// SIMATIC S7-200 project (STEP 7-Micro/WIN), CPU 222 REL 02.01

SYMBOL_TABLE USER1
AI_1             AIW0     // TEMPERATURA DI SERVIZIO O RICIRCOLO
AI_2             AIW2     // TEMPERATURA CALDAIA
AI_3             AIW4     // TEMPERATURA AMBIENTE
AI_4             AIW6     // TEMPERATURA CIRCUITO DI RITORNO
M                AQW0     // COMANDO VALVOLA DI MISCELAZIONE
B1               Q0.0     // POMPA DI CIRCOLAZIONE LIVELLO 1
B2               Q0.1     // POMPA DI CIRCOLAZIONE LIVELLO 2
B3               Q0.2     // POMPA DI CIRCOLAZIONE LIVELLO 3
POMPA_2          Q0.3     // POMPA RISCALDAMENTO ACQUA USO DOMESTICO
BRC_1            Q0.4     // BRUCCIATORE LIVELLO 1
BRC_2            Q0.5     // BRUCCIATORE LIVELLO 2
BRC_3            Q1.0     // BRUCCIATORE LIVELLO 3
MIS_T_SERV       VD0      // MISURA TEMPERATURA DI SERVIZIO
MIS_T_CALDAIA    VD4      // MISURA TEMPERATURA CALDAIA
MIS_T_AMBIENTE   VD8      // MISURA TEMPERATURA AMBIENTE
MIS_T_RIT        VD12     // MISURA TEMPERATURA DI RITORNO
D_T              VD16     // DIFFERENZA DI TEMPERATURA FRA CALDAIA E RITORNO
END_SYMBOL_TABLE

ORGANIZATION_BLOCK MAIN:OB1
TITLE=DPS 210 IMPIANTO DI RISCALDAMENTO
BEGIN
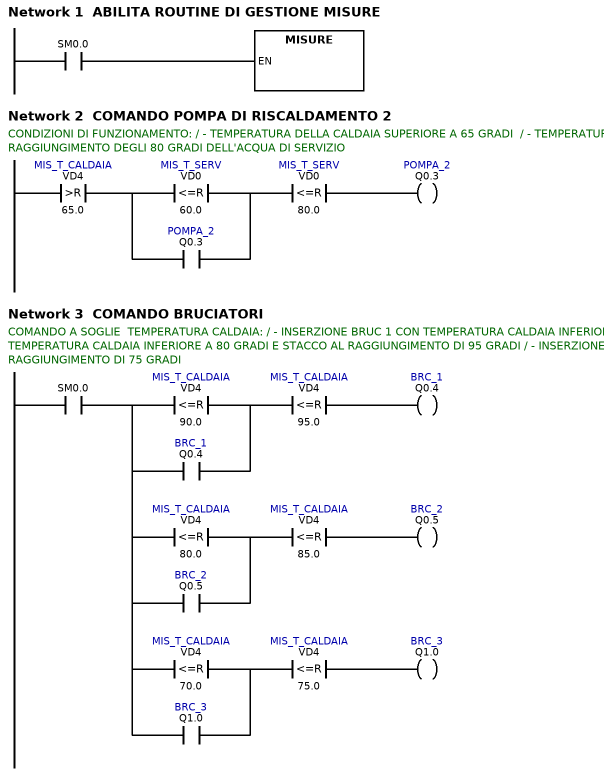
Network 1 // ABILITA ROUTINE DI GESTIONE MISURE
LD     SM0.0
CALL   MISURE:SBR1
Network 2 // COMANDO POMPA DI RISCALDAMENTO 2
// CONDIZIONI DI FUNZIONAMENTO:
// - TEMPERATURA DELLA CALDAIA SUPERIORE A 65 GRADI 
// - TEMPERATURA DI SERVIZIO INFERIORE A 60 GRADI
// PARTE LA POMPA DI CIRCOLAZIONE 2 FINO AL RAGGIUNGIMENTO DEGLI 80 GRADI DELL'ACQUA DI SERVIZIO
LDR>   MIS_T_CALDAIA:VD4, 65.0
LDR<=  MIS_T_SERV:VD0, 60.0
O      POMPA_2:Q0.3
ALD
AR<=   MIS_T_SERV:VD0, 80.0
=      POMPA_2:Q0.3
Network 3 // COMANDO BRUCIATORI
// COMANDO A SOGLIE  TEMPERATURA CALDAIA:
// - INSERZIONE BRUC 1 CON TEMPERATURA CALDAIA INFERIORE A 90 GRADI E STACCO AL RAGGIUNGIMENTO DI 95 GRADI
// - INSERZIONE BRUC 2 CON TEMPERATURA CALDAIA INFERIORE A 80 GRADI E STACCO AL RAGGIUNGIMENTO DI 95 GRADI
// - INSERZIONE BRUC 3 CON TEMPERATURA CALDAIA INFERIORE A 70 GRADI E STACCO AL RAGGIUNGIMENTO DI 75 GRADI
LD     SM0.0
LPS
LDR<=  MIS_T_CALDAIA:VD4, 90.0
O      BRC_1:Q0.4
ALD
AR<=   MIS_T_CALDAIA:VD4, 95.0
=      BRC_1:Q0.4
LRD
LDR<=  MIS_T_CALDAIA:VD4, 80.0
O      BRC_2:Q0.5
ALD
AR<=   MIS_T_CALDAIA:VD4, 85.0
=      BRC_2:Q0.5
LPP
LDR<=  MIS_T_CALDAIA:VD4, 70.0
O      BRC_3:Q1.0
ALD
AR<=   MIS_T_CALDAIA:VD4, 75.0
=      BRC_3:Q1.0
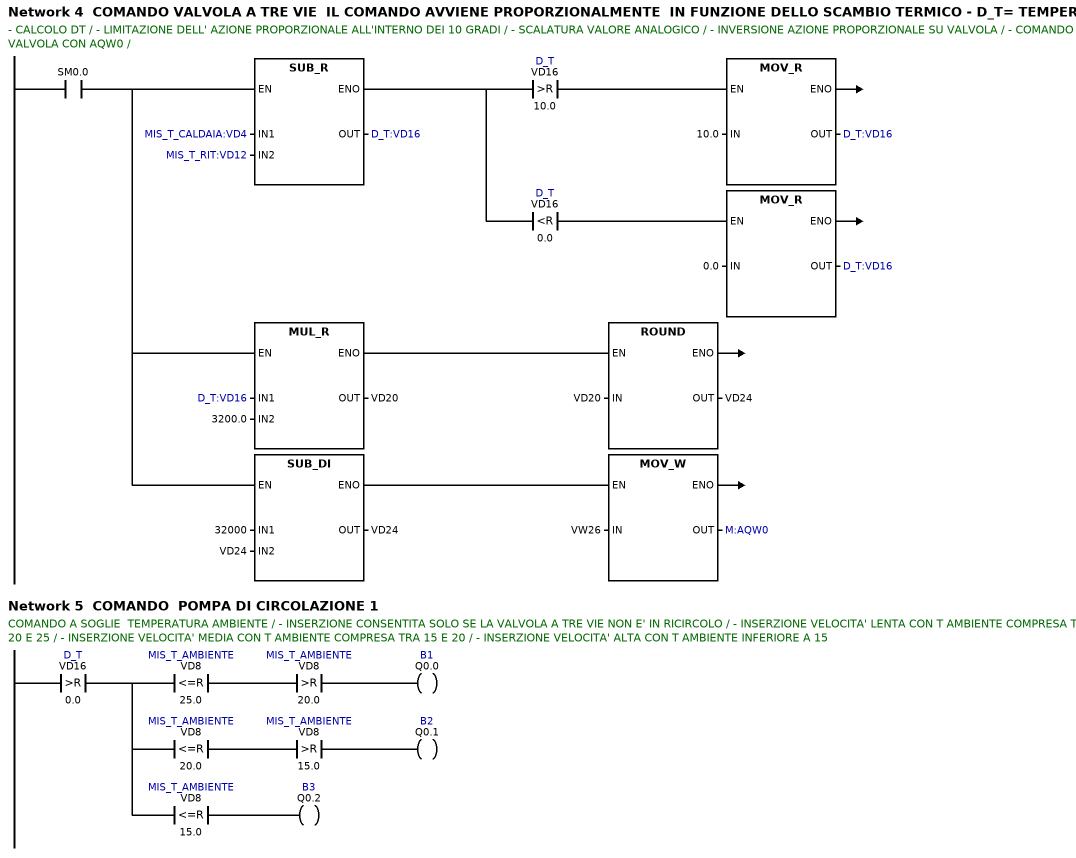
Network 4 // COMANDO VALVOLA A TRE VIE 
IL COMANDO AVVIENE PROPORZIONALMENTE  IN FUNZIONE DELLO SCAMBIO TERMICO
- D_T= TEMPERATURA CALDAIA - TEMPERATURA RITORNO
- D_T =0 VALVOLA TRE VIE IN RICIRCOLO
- D_T= 10 VALVOLA TRE VIE IN PIENA MANDATA
// - CALCOLO DT
// - LIMITAZIONE DELL' AZIONE PROPORZIONALE ALL'INTERNO DEI 10 GRADI
// - SCALATURA VALORE ANALOGICO
// - INVERSIONE AZIONE PROPORZIONALE SU VALVOLA
// - COMANDO VALVOLA CON AQW0
// 
LD     SM0.0
LPS
MOVR   MIS_T_CALDAIA:VD4, D_T:VD16
AENO
-R     MIS_T_RIT:VD12, D_T:VD16
AENO
LPS
AR>    D_T:VD16, 10.0
MOVR   10.0, D_T:VD16
LPP
AR<    D_T:VD16, 0.0
MOVR   0.0, D_T:VD16
LPP
LPS
MOVR   D_T:VD16, VD20
AENO
*R     3200.0, VD20
AENO
ROUND  VD20, VD24
LPP
INVD   VD24
AENO
INCD   VD24
AENO
+D     32000, VD24
AENO
MOVW   VW26, M:AQW0
Network 5 // COMANDO  POMPA DI CIRCOLAZIONE 1
// COMANDO A SOGLIE  TEMPERATURA AMBIENTE
// - INSERZIONE CONSENTITA SOLO SE LA VALVOLA A TRE VIE NON E' IN RICIRCOLO
// - INSERZIONE VELOCITA' LENTA CON T AMBIENTE COMPRESA TRA 20 E 25
// - INSERZIONE VELOCITA' MEDIA CON T AMBIENTE COMPRESA TRA 15 E 20
// - INSERZIONE VELOCITA' ALTA CON T AMBIENTE INFERIORE A 15
LDR>   D_T:VD16, 0.0
LPS
AR<=   MIS_T_AMBIENTE:VD8, 25.0
AR>    MIS_T_AMBIENTE:VD8, 20.0
=      B1:Q0.0
LRD
AR<=   MIS_T_AMBIENTE:VD8, 20.0
AR>    MIS_T_AMBIENTE:VD8, 15.0
=      B2:Q0.1
LPP
AR<=   MIS_T_AMBIENTE:VD8, 15.0
=      B3:Q0.2
END_ORGANIZATION_BLOCK

SUBROUTINE_BLOCK SCALA:SBR0
TITLE=COMMENTI SUL SOTTOPROGRAMMA
VAR_INPUT
x:WORD;	// LW0 
x1:REAL;	// LD2 
x2:REAL;	// LD6 
y1:REAL;	// LD10 
y2:REAL;	// LD14 
END_VAR
VAR_OUTPUT
y:REAL;	// LD18 
END_VAR
BEGIN
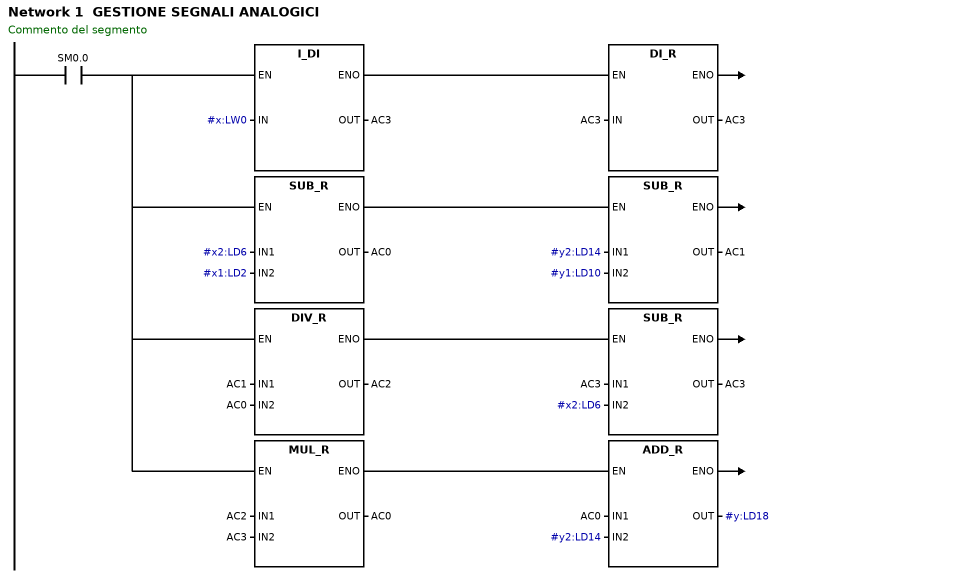
Network 1 // GESTIONE SEGNALI ANALOGICI
// Commento del segmento
LD     SM0.0
LPS
ITD    #x:LW0, AC3
AENO
DTR    AC3, AC3
LRD
MOVR   #x2:LD6, AC0
AENO
-R     #x1:LD2, AC0
AENO
MOVR   #y2:LD14, AC1
-R     #y1:LD10, AC1
LRD
MOVR   AC1, AC2
AENO
/R     AC0, AC2
AENO
-R     #x2:LD6, AC3
LPP
MOVR   AC2, AC0
AENO
*R     AC3, AC0
AENO
MOVR   AC0, #y:LD18
+R     #y2:LD14, #y:LD18
Network 2 // Titolo del segmento
// Commento del segmento
END_SUBROUTINE_BLOCK

SUBROUTINE_BLOCK MISURE:SBR1
TITLE=SCALA GLI INGRESSI ANALOGICI DA 0-100
BEGIN
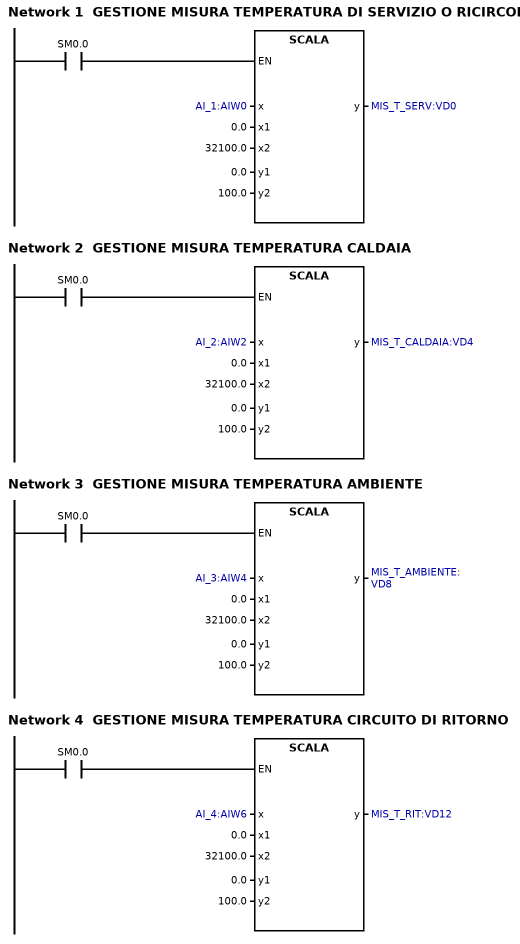
Network 1 // GESTIONE MISURA TEMPERATURA DI SERVIZIO O RICIRCOLO
LD     SM0.0
CALL   SCALA:SBR0, AI_1:AIW0, 0.0, 32100.0, 0.0, 100.0, MIS_T_SERV:VD0
Network 2 // GESTIONE MISURA TEMPERATURA CALDAIA
LD     SM0.0
CALL   SCALA:SBR0, AI_2:AIW2, 0.0, 32100.0, 0.0, 100.0, MIS_T_CALDAIA:VD4
Network 3 // GESTIONE MISURA TEMPERATURA AMBIENTE
LD     SM0.0
CALL   SCALA:SBR0, AI_3:AIW4, 0.0, 32100.0, 0.0, 100.0, MIS_T_AMBIENTE:VD8
Network 4 // GESTIONE MISURA TEMPERATURA CIRCUITO DI RITORNO
LD     SM0.0
CALL   SCALA:SBR0, AI_4:AIW6, 0.0, 32100.0, 0.0, 100.0, MIS_T_RIT:VD12
Network 5 // Titolo del segmento
// Commento del segmento
END_SUBROUTINE_BLOCK
